(* CoDeSys 2.3 export: PLC_PRG.EXP *)

(* POU PLC_PRG, ST *)
PROGRAM PLC_PRG
VAR CONSTANT
	K14AutoModeDelay : TIME := T#10s;
END_VAR

VAR
	SignalizationResetTrigger : R_TRIG;
	K14PumpsControl : fbK14PumpsControl;
	K15PumpsControl : fbK15PumpsControl;
	K16PumpsControl : fbK16PumpsControl;
	K14ManualModeTOF : TOF;
END_VAR

VAR_TEMP
	i: USINT;
	turnOnK14PumpButtonPressed : ARRAY [1..MAX_K14_PUMPS_NUM] OF BOOL;
	turnOffK14PumpButtonPressed : ARRAY [1..MAX_K14_PUMPS_NUM] OF BOOL;
	emergencyK14PumpStopButtonPressed : ARRAY [1..MAX_K14_PUMPS_NUM] OF BOOL;
	K14PumpState : ARRAY [1..MAX_K14_PUMPS_NUM] OF BOOL;
	K14WorkAllowed : BOOL := FALSE;


	turnOnK15PumpButtonPressed : ARRAY [1..MAX_K15_PUMPS_NUM] OF BOOL;
	turnOffK15PumpButtonPressed : ARRAY [1..MAX_K15_PUMPS_NUM] OF BOOL;
	emergencyK15PumpStopButtonPressed : ARRAY [1..MAX_K15_PUMPS_NUM] OF BOOL;
	K15PumpState : ARRAY [1..MAX_K15_PUMPS_NUM] OF BOOL;
	K15WorkAllowed: BOOL := FALSE;

	turnOnK16PumpButtonPressed : ARRAY [1..MAX_K16_PUMPS_NUM] OF BOOL;
	turnOffK16PumpButtonPressed : ARRAY [1..MAX_K16_PUMPS_NUM] OF BOOL;
	emergencyK16PumpStopButtonPressed : ARRAY [1..MAX_K16_PUMPS_NUM] OF BOOL;
	K16PumpState : ARRAY [1..MAX_K16_PUMPS_NUM] OF BOOL;
	K16WorkAllowed : BOOL := FALSE;
END_VAR
(*
	Сброс всех аварий насосов по замыканию кнопки
	съема аварий
*)
SignalizationResetTrigger(CLK := MV110DI.SignalizationButton);
resetPumpsAlarm(SignalizationResetTrigger.Q);


(*
	Включение сигнала на UZ
	по тому же сигналу, что и MV110DI.TurnOnK15AndK16
*)
FOR i := 1 TO MAX_K14_PUMPS_NUM DO
	PLC160DO.UZStart[i] := MV110DI.TurnOnK15AndK16;
END_FOR;

(*
	3. Управление насосами К14
	контура отопления и вентиляции
*)
FOR i := 1 TO MAX_K14_PUMPS_NUM DO
	turnOnK14PumpButtonPressed[i] := NOT(PLC160DI.K14_PumpStop[i]);
	turnOffK14PumpButtonPressed[i] := PLC160DI.K14_PumpStop[i];
	emergencyK14PumpStopButtonPressed[i] := PLC160DI.UZStatus[i].Fail;

	MU110DO.K14PumpIsOn[i] := PLC160DI.UZStatus[i].Running;
	(*Включить/Выключить сигнальную лампу состояния насоса*)

	K14PumpState[i] := MU110DO.K14PumpIsOn[i];

	(*если хоть один из насосов исправен, то работа разрешена*)
	IF NOT(K14PumpFaulty[i]) THEN
		K14WorkAllowed := TRUE;
	END_IF;
END_FOR;

K14ManualModeTOF(IN := NOT(PLC160DI.K14_PumpsModeIsAuto), PT := K14AutoModeDelay);

K14PumpsControl(
	ManualMode						:= K14ManualModeTOF.Q,
	WorkAllowed						:= K14WorkAllowed,
	SummerMode						:= NOT(PLC160DI.K14_PumpsModeIsHeating),
	TurnOnPumpButtonPressed		:= turnOnK14PumpButtonPressed, (*TODO: Выяснить про этот вход*)
	TurnOffPumpButtonPressed	:= turnOffK14PumpButtonPressed,
	EmergencyPumpStopButtonPressed := emergencyK14PumpStopButtonPressed,		(*TODO: Выяснить про этот вход*)
	PumpState						:= K14PumpState,
	PressureDrop					:= NOT(PLC160DI.K14_NoPressureDrop)
);

(*
	6. Управление насосами К15
	греющего контура ГВС
*)
FOR i := 1 TO MAX_K15_PUMPS_NUM DO
	turnOnK15PumpButtonPressed[i] := NOT(MV110DI.K15_StopButton[i]);
	turnOffK15PumpButtonPressed[i] := MV110DI.K15_StopButton[i];
	emergencyK15PumpStopButtonPressed[i] := FALSE;
	K15PumpState[i] := PLC160DO.K15Pump[i];
	(*если хоть один из насосов исправен, то работа разрешена*)
	IF NOT(K15PumpFaulty[i]) THEN
		K15WorkAllowed := TRUE;
	END_IF;
END_FOR;

K15PumpsControl(
	ManualMode						:= NOT(MV110DI.HeatingDHWPumpGroupModeIsAuto),
	WorkAllowed						:= K15WorkAllowed,
	TurnOnPumpButtonPressed		:= turnOnK15PumpButtonPressed, (*TODO: Выяснить про этот вход*)
	TurnOffPumpButtonPressed	:= turnOffK15PumpButtonPressed,
	EmergencyPumpStopButtonPressed := emergencyK15PumpStopButtonPressed,		(*TODO: Выяснить про этот вход*)
	PumpState						:= K15PumpState,
	PressureDrop					:= NOT(MV110DI.K15_NoPressureDrop)
);

(*
	5. Управление насосами К16
	контура ГВС
*)
FOR i := 1 TO MAX_K16_PUMPS_NUM DO
	turnOnK16PumpButtonPressed[i] := NOT(MV110DI.K16_StopButton[i]);
	turnOffK16PumpButtonPressed[i] := MV110DI.K16_StopButton[i];
	emergencyK16PumpStopButtonPressed[i] := FALSE;
	K16PumpState[i] := PLC160DO.K16Pump[i];

	(*если хоть один из насосов исправен, то работа разрешена*)
	IF NOT(K16PumpFaulty[i]) THEN
		K16WorkAllowed := TRUE;
	END_IF;
END_FOR;

K16PumpsControl(
	ManualMode						:= NOT(MV110DI.DHWPumpGroupModeIsAuto),
	WorkAllowed						:= K16WorkAllowed,
	TurnOnPumpButtonPressed		:= turnOnK16PumpButtonPressed, (*TODO: Выяснить про этот вход*)
	TurnOffPumpButtonPressed	:= turnOffK16PumpButtonPressed,
	EmergencyPumpStopButtonPressed := emergencyK16PumpStopButtonPressed,		(*TODO: Выяснить про этот вход*)
	PumpState						:= K16PumpState,
	PressureDrop					:= NOT(MV110DI.K16_NoPressureDrop)
);
END_PROGRAM
